Staubli VAL3: defineTraj.pgx

program defineTraj()
  local num i
  local num l_nType
  local string l_sPath
begin
//  // select the trajectory type
//  if saveData:sTrajTypeUsing==""
//    saveData:sTrajTypeUsing=saveData:sTrajType
//  endIf
//  // search inside all the instruction
//  call saveData:getPathInstr(saveData:sTrajTypeUsing,l_sPath)
//  // check the trajType
//  if trajType:libPath()!=l_sPath and l_sPath!=""
//    i=trajType:libLoad(l_sPath)
//    delay(0)
//  endIf
//  // error
//  if i!=0
//    popUpMsg("error load traj type on ENTER"+saveData:sTrajTypeUsing+toString("",i))
//  endIf
end
